(* IEC 61131-3 sources: LLM-CodeGen-TestGen/Tests, 13 files *)

(* ---- CRC_GEN.st ---- *)
FUNCTION_BLOCK CRC_GEN
  VAR_IN_OUT
    PT : ARRAY [0..249] OF BYTE;
  END_VAR
  VAR_INPUT
    SIZE : UINT;
    PL : UINT;
    PN : DWORD;
    INIT : DWORD;
    REV_IN : BOOL;
    REV_OUT : BOOL;
    XOR_OUT : DWORD;
  END_VAR
  VAR_OUTPUT
    _CRC_GEN : DWORD;
  END_VAR
  VAR
    pos : INT;
    shift : INT;
    bits : INT;
    dx : BYTE;
  END_VAR

  shift := 32 - UINT_TO_INT(PL);
  PN := SHL(PN, shift);

  (* load first 4 bytes into register minimum message size is 4 bytes
  	for smaller messages fill with 0#s at the beginning*)
  FOR pos := 0 TO 3 DO
  	IF REV_IN THEN _CRC_GEN := SHL(_CRC_GEN, 8) OR BYTE_TO_DWORD(REVERSE(PT[pos])); ELSE _CRC_GEN := SHL(_CRC_GEN, 8) OR BYTE_TO_DWORD(PT[pos]); END_IF;
  END_FOR;
  pos := 4;

  (* xor with init value *)
  _CRC_GEN := _CRC_GEN XOR SHL(init, shift);

  (* calculate CRC for each byte *)
  WHILE pos < UINT_TO_INT(size) DO
  	IF REV_IN THEN DX := REVERSE(PT[pos]); ELSE DX := PT[pos]; END_IF;
  	pos := pos + 1;
  	(* crc calculation for one byte *)
  	FOR bits := 0 TO 7 DO
  		IF (_CRC_GEN AND DWORD#16#8000_0000) > DWORD#0 THEN (* CRC_GEN.31 *)
  			_CRC_GEN := (SHL(_CRC_GEN, 1) OR BOOL_TO_DWORD((DX AND BYTE#16#80) > BYTE#0)) XOR PN; (* DX.7 *)
  		ELSE
  			_CRC_GEN := SHL(_CRC_GEN, 1) OR BOOL_TO_DWORD((DX AND BYTE#16#80) > BYTE#0); (* DX.7 *)
  		END_IF;
  		dx := SHL(dx, 1);
  	END_FOR;
  END_WHILE;

  (* all bytes are processed, need to finish the registers 32 bits *)
  FOR bits := 0 TO 31 DO
  	IF (_CRC_GEN AND DWORD#16#8000_0000) > DWORD#0 THEN (* CRC_GEN.31 *)
  		_CRC_GEN := (SHL(_CRC_GEN, 1) OR BOOL_TO_DWORD((DX AND BYTE#16#80) > BYTE#0)) XOR PN; (* DX.7 *)
  	ELSE
  		_CRC_GEN := SHL(_CRC_GEN, 1) OR BOOL_TO_DWORD((DX AND BYTE#16#80) > BYTE#0); (* DX.7 *)
  	END_IF;
  END_FOR;

  (* final XOR *)
  _CRC_GEN := SHR(_CRC_GEN, shift) XOR XOR_OUT;

  (* reverse the crc_out put if necessary *)
  IF REV_OUT THEN _CRC_GEN := REFLECT(_CRC_GEN, UINT_TO_INT(PL)); END_IF;

  (* typical crc polynoms

  CRC-4-ITU 			x4 + x + 1 					(ITU G.704, p. 12) 	0x3 or 0xC (0x9)
  CRC-5-ITU 			x5 + x4 + x2 + 1 			(ITU G.704, p. 9) 	0x15 or 0x15 (0x0B) Bluetooth
  CRC-5-USB 			x5 + x2 + 1 				(use: USB token packets) 	0x05 or 0x14 (0x9)
  CRC-6-ITU 			x6 + x + 1 					(ITU G.704, p. 3) 	0x03 or 0x30 (0x21)
  CRC-7 				x7 + x3 + 1 				(use: telecom systems, MMC) 	0x09 or 0x48 (0x11)
  CRC-8-ATM 			x8 + x2 + x + 1 				(use: ATM HEC) 	0x07 or 0xE0 (0xC1)
  CRC-8-CCITT 		x8 + x7 + x3 + x2 + 1 		(use: 1-Wire bus) 	0x8D or 0xB1 (0x63)
  CRC-8-Dallas/Maxim 	x8 + x5 + x4 + 1 			(use: 1-Wire bus) 	0x31 or 0x8C (0x19)
  CRC-8 				x8 + x7 + x6 + x4 + x2 + 1 	0xD5 or 0xAB (0x57)
  CRC-8-SAE J1850 	x8 + x4 + x3 + x2 + 1 		0x1D or 0xB8
  CRC-10 				x10 + x9 + x5 + x4 + x + 1 	0x233 or 0x331 (0x263)
  CRC-12 				x12 + x11 + x3 + x2 + x + 1 (use: telecom systems) 	0x80F or 0xF01 (0xE03)
  CRC-15-CAN 			x15 + x14 + x10 + x8 + x7 + x4 + x3 + 1 	0x4599 or 0x4CD1 (0x19A3)
  CRC-16-Fletcher 	Not a CRC; see Fletchers checksum 	Used in Adler-32 A & B CRCs
  CRC-16-CCITT 	x16 + x12 + x5 + 1 (XMODEM,X.25, V.41, Bluetooth, PPP, IrDA; known as "CRC-CCITT") 	0x1021 or 0x8408 (0x0811)
  CRC-16-IBM 	x16 + x15 + x2 + 1 (USB, many others; also known as "CRC-16") 	0x8005 or 0xA001 (0x4003)
  CRC-24-Radix-64 	x24 + x23 + x18 + x17 + x14 + x11 + x10 + x7 + x6 + x5 + x4 + x3 + x + 1 	0x864CFB or 0xDF3261 (0xBE64C3)
  CRC-32-Adler 	Not a CRC; see Adler-32 	See Adler-32
  CRC-32-MPEG2 	x32 + x26 + x23 + x22 + x16 + x12 + x11 + x10 + x8 + x7 + x5 + x4 + x2 + x + 1 	0x04C11DB7 or 0xEDB88320 (0xDB710641) Also used in IEEE 802.3
  CRC-32-IEEE 802.3 	x32 + x26 + x23 + x22 + x16 + x12 + x11 + x10 + x8 + x7 + x5 + x4 + x2 + x + 1 (V.42) 	0x04C11DB7 or 0xEDB88320 (0xDB710641)
  CRC-32C (Castagnoli) 	x32 + x28 + x27 + x26 + x25 + x23 + x22 + x20 + x19 + x18 + x14 + x13 + x11 + x10 + x9 + x8 + x6 + 1 	0x1EDC6F41 or 0x82F63B78 (0x05EC76F1)
  CRC-64-ISO 	x64 + x4 + x3 + x + 1 (use: ISO 3309) 	0x000000000000001B or 0xD800000000000000 (0xB000000000000001)
  CRC-64-ECMA-182 	x64 + x62 + x57 + x55 + x54 + x53 + x52 + x47 + x46 + x45 + x40 + x39 + x38 + x37 + x35 + x33 + x32 + x31 + x29 + x27 + x24 + x23 + x22 + x21 + x19 + x17 + x13 + x12 + x10 + x9 + x7 + x4 + x + 1
  (as described in ECMA-182 p.63) 	0x42F0E1EBA9EA3693 or 0xC96C5795D7870F42 (0x92D8AF2BAF0E1E85)
  *)
END_FUNCTION_BLOCK

(* ---- DEC_TO_HEX.st ---- *)
FUNCTION_BLOCK DEC_TO_HEX
  VAR_INPUT
    DecimalValue : DINT;
  END_VAR
  VAR_OUTPUT
    HexString : STRING;
  END_VAR
  VAR
    i : INT;
    hexDigits : ARRAY [0..15] OF STRING := ['0', '1', '2', '3', '4', '5', '6', '7', '8', '9', 'A', 'B', 'C', 'D', 'E', 'F'];
    digitIndex : INT;
    hexDigit : STRING;
    significantDigitFound : BOOL := FALSE;
    digitValue : DINT;
    powerOfInteger : DINT;
  END_VAR

  HexString := '';

  IF DecimalValue = 0 THEN
      HexString := '0';
      RETURN;
  END_IF;

  significantDigitFound := FALSE;

  FOR digitIndex := 0 TO 7 DO

      powerOfInteger:=1;
      FOR i := 1 TO 7 - digitIndex DO
        powerOfInteger := powerOfInteger * 16;
      END_FOR;

      digitValue := DIV(DecimalValue, powerOfInteger) MOD 16;
      hexDigit := hexDigits[digitValue];

      IF hexDigit <> '0' OR significantDigitFound OR (7 - digitIndex) = 0 THEN
          significantDigitFound := TRUE;
          HexString := CONCAT(HexString, hexDigit);
      END_IF;

  END_FOR;
END_FUNCTION_BLOCK

(* ---- FLOW_METER.st ---- *)
FUNCTION_BLOCK FLOW_METER
  VAR_INPUT
    VX : REAL;
    _E : BOOL;
    RST : BOOL;
    PULSE_MODE : BOOL;
    UPDATE_TIME : TIME := t#1s;
  END_VAR
  VAR_OUTPUT
    F : REAL;
  END_VAR
  VAR_IN_OUT
    X : REAL;
    Y : UDINT;
  END_VAR
  VAR
    tx : TIME;
    tl : TIME;
    int1 : INTEGRATE;
    init : BOOL;
    e_last : BOOL;
    tmp : INT;
    x_last : REAL;
    y_last : UDINT;
  END_VAR

  IF NOT init THEN	(* init on power up *)
  	init := TRUE;
  	tl := tx;
  	x_last := X;
  	y_last := Y;
  	int1.K := 2.7777777777777777E-4;
  END_IF;

  (* run integrator *)
  int1(_E := NOT (RST OR PULSE_MODE) AND _E, X := VX, Y := X);	(* gated operation *)
  X := int1.Y;

  IF RST THEN		(* reset *)
  	X := 0.0;
  	Y := UDINT#0;
  	tl := tx;
  	x_last := 0.0;
  	y_last := UDINT#0;
  ELSIF _E AND PULSE_MODE THEN	(* check for pulse mode *)
  	IF NOT e_last THEN X := X + VX; END_IF;
  END_IF;
  e_last := _E;

  (* reduce X to be less than 1 and increase Y respectively *)
  IF X > 1.0 THEN
  	tmp := FLOOR(X);
  	Y := Y + INT_TO_UDINT(tmp);
  	X := X - INT_TO_REAL(tmp);
  END_IF;

  (* calculate the current flow *)
  tx := UDINT_TO_TIME(T_PLC_MS(en:=true));
  IF tx - tl >= UPDATE_TIME AND UPDATE_TIME > t#0s THEN
  	F := (UDINT_TO_REAL(Y - y_last) + X - x_last) / TIME_TO_REAL(tx - tl) * 3.6E6;
  	y_last := Y;
  	x_last := X;
  	tl := tx;
  END_IF;

  (* From OSCAT Library, www.oscat.de *)
  (* T_PLC_MS, FLOOR, INTEGRATE required *)
END_FUNCTION_BLOCK

(* ---- FT_PIDWL.st ---- *)
FUNCTION_BLOCK FT_PIDWL
  VAR_INPUT
    IN : REAL;
    KP : REAL := 1.0;
    TN : REAL := 1.0;
    TV : REAL := 1.0;
    LIM_L : REAL := -1.0E38;
    LIM_H : REAL := 1.0E38;
    RST : BOOL;
  END_VAR
  VAR_OUTPUT
    Y : REAL;
    LIM : BOOL;
  END_VAR
  VAR
    piwl : FT_PIWL;
    diff : FT_DERIV;
  END_VAR

  IF rst THEN
  	piwl(rst := TRUE);
  	piwl.RST := FALSE;
  ELSE
  	(* run PIWL controller first *)
  	(* we need to check if TN = 0 and do alternative calls *)
  	IF TN = 0.0 THEN
  		piwl(in := IN * KP, KP := 1.0, KI := 0.0, LIM_L := LIM_L, LIM_H := LIM_H);
  	ELSE
  		piwl(in := IN * KP, KP := 1.0, KI := 1.0 / TN, LIM_L := LIM_L, LIM_H := LIM_H);
  	END_IF;

  	(* run differentiator and add_to_output *)
  	diff(IN := IN, K := KP * TV);
  	Y := piwl.Y + diff.out;

  	(* limit the output *)
  	IF Y < LIM_L THEN
  		LIM := TRUE;
  		Y := LIM_L;
  	ELSIF Y > LIM_H THEN
  		LIM := TRUE;
  		Y := LIM_H;
  	ELSE
  		LIM := FALSE;
  	END_IF;
  END_IF;

  (* From OSCAT Library, www.oscat.de *)
  (* T_PLC_US, FT_DERIV required *)
END_FUNCTION_BLOCK

(* ---- GEN_BIT.st ---- *)
FUNCTION_BLOCK GEN_BIT
  VAR_INPUT
    IN0 : DWORD;
    IN1 : DWORD;
    IN2 : DWORD;
    IN3 : DWORD;
    CLK : BOOL;
    STEPS : INT;
    REP : INT;
    RST : BOOL;
  END_VAR
  VAR_OUTPUT
    Q0 : BOOL;
    Q1 : BOOL;
    Q2 : BOOL;
    Q3 : BOOL;
    CNT : INT;
    RUN : BOOL;
  END_VAR
  VAR
    r0 : DWORD;
    r1 : DWORD;
    r2 : DWORD;
    r3 : DWORD;
    rx : INT := 1;
  END_VAR

  (* check if number of runs is finished or rep = 0 which means continuous *)

  IF clk AND NOT rst THEN
  	run := (rep = 0) OR (rx <= rep);
  	IF run THEN
  		(* check for step counter reached and reset to 0 if cnt = steps *)
  		IF cnt = steps THEN
  			cnt := 0;
  		END_IF;

  		(* when cnt = 0 then reload the inputs into the registers *)
  		IF cnt = 0 THEN
  			r0 := in0;
  			r1 := in1;
  			r2 := in2;
  			r3 := in3;
  		END_IF;

  		(* when cnt < steps, shift the lowest bits to the outputs *)
  		IF (cnt < steps) THEN
              Q0 := BIT_OF_DWORD(r0,0); (* Q0 := r0.X0; *)
              Q1 := BIT_OF_DWORD(r1,0); (* Q1 := r1.X0; *)
              Q2 := BIT_OF_DWORD(r2,0); (* Q2 := r2.X0; *)
              Q3 := BIT_OF_DWORD(r3,0); (* Q3 := r3.X0; *)
  			r0 := SHR(r0,1);
  			r1 := SHR(r1,1);
  			r2 := SHR(r2,1);
  			r3 := SHR(r3,1);
  		END_IF;

  		(* increment the step counter *)
  		cnt := cnt +1;
  		IF (cnt = steps) AND (rep <> 0) THEN rx := rx +1; END_IF;
  		IF (rx > rep) AND (rep <> 0) THEN run := FALSE; END_IF;
  	END_IF;
  ELSE
  	IF rst THEN
  		run := FALSE;
  		Q0 := FALSE;
  		Q1 := FALSE;
  		Q2 := FALSE;
  		Q3 := FALSE;
  		r0 := DWORD#0;
  		r1 := DWORD#0;
  		r2 := DWORD#0;
  		r3 := DWORD#0;
  		cnt := 0;
  		rx := 1;
  	END_IF;
  END_IF;

  (*From OSCAT Library, www.oscat.de *)
END_FUNCTION_BLOCK

(* ---- GEN_SIN.st ---- *)
FUNCTION_BLOCK GEN_SIN
  VAR_INPUT
    PT : TIME;
    AM : REAL := 1.0;
    OS : REAL;
    DL : REAL;
  END_VAR
  VAR_OUTPUT
    Q : BOOL;
    OUT : REAL;
  END_VAR
  VAR
    tx : TIME;
    last : TIME;
    init : BOOL;
    temp : REAL;
  END_VAR

  tx:= UDINT_TO_TIME(T_PLC_MS(en:=true)) - last;

  DL := modR(dl,1.0);
  IF dl < 0.0 THEN dl := 1.0 - dl; END_IF;

  (* init section *)
  IF NOT init THEN
  	init := TRUE;
  	last := tx;
  	tx := t#0s;
  END_IF;

  (* add last if one cycle is finished *)
  IF tx >= pt THEN
  	last := last + pt;
  	tx := tx - pt;
  END_IF;

  (* generate sine wave *)
  IF pt > t#0s THEN temp := SIN(6.283185307179586476 * TIME_TO_REAL(tx + multime(pt, dl)) / TIME_TO_REAL(pt)); END_IF;
  out := am * 0.5 *  temp + os;

  (* boolean output Q *)
  q := NOT sign_R(temp);

  (* From OSCAT Library, www.oscat.de *)
  (* T_PLC_MS, SIGN_R required*)
END_FUNCTION_BLOCK

(* ---- INCLUDE.st ---- *)
FUNCTION BIT_OF_DWORD : BOOL
  VAR_INPUT
    IN : DWORD;
    N : INT;
  END_VAR

  BIT_OF_DWORD := (SHR(in,N) AND 16#00000001) > 0;
  (* from OSCAT library; www.oscat.de  *)
END_FUNCTION

FUNCTION SIGN_R : BOOL
  VAR_INPUT
    IN : REAL;
  END_VAR

  SIGN_R := in < 0.0;
  (* from OSCAT library; www.oscat.de  *)
END_FUNCTION

FUNCTION FLOOR : INT
  VAR_INPUT
    x : REAL;
  END_VAR

  FLOOR := REAL_TO_INT(X);
  IF INT_TO_REAL(FLOOR) > X THEN
  	floor := floor - 1;
  END_IF;
  (* from OSCAT library; www.oscat.de  *)
END_FUNCTION

FUNCTION FLOOR2 : DINT
  VAR_INPUT
    x : REAL;
  END_VAR

  FLOOR2 := REAL_TO_DINT(X);
  IF DINT_TO_REAL(FLOOR2) > X THEN
  	FLOOR2 := FLOOR2 - DINT#1;
  END_IF;
  (* from OSCAT library; www.oscat.de  *)
END_FUNCTION

FUNCTION MODR : REAL
  VAR_INPUT
    IN : REAL;
    DIVI : REAL;
  END_VAR

  IF divi = 0.0 THEN
  	MODR := 0.0;
  ELSE
  	MODR := in - DINT_TO_REAL(FLOOR2(in / divi)) * divi;
  END_IF;
  (* from OSCAT library; www.oscat.de  *)
  (* FC FLOOR2 required *)
END_FUNCTION

FUNCTION REVERSE : BYTE
  VAR_INPUT
    IN : BYTE;
  END_VAR

  reverse := SHL(in,7) OR SHR(in,7) OR (ROR(in,3) AND BYTE#2#01000100) OR (ROL(in,3) AND BYTE#2#00100010)
  	OR (SHL(in,1) AND BYTE#2#00010000) OR (SHR(in,1) AND BYTE#2#00001000);

  (* Fromm Oscat Library, www.oscat.de *)
END_FUNCTION

FUNCTION REFLECT : DWORD
  VAR_INPUT
    DI : DWORD;
    L : INT;
  END_VAR
  VAR
    i : INT;
    _d : DWORD;
  END_VAR

  _d := DI;
  FOR i := 1 TO L DO
  	REFLECT := SHL(REFLECT, 1) OR BOOL_TO_DWORD((_d AND DWORD#2#0000_0001) > DWORD#0); (* D.0 *)
  	_d := SHR(_d, 1);
  END_FOR;
  REFLECT := REFLECT OR SHL(_d, L);

  (* Fromm Oscat Library, www.oscat.de *)
END_FUNCTION

FUNCTION BIT_LOAD_B : BYTE
  VAR_INPUT
    IN : BYTE;
    VAL : BOOL;
    POS : INT;
  END_VAR

  IF VAL THEN
  	BIT_LOAD_B := in OR SHL(BYTE#1,pos);
  ELSE
  	BIT_LOAD_B := in AND (NOT SHL(BYTE#1,pos));
  END_IF;

  (*From OSCAT Library, www.oscat.de*)
END_FUNCTION

FUNCTION _BYTE_TO_INT : INT
  VAR_INPUT
    IN : BYTE;
  END_VAR

  _BYTE_TO_INT := USINT_TO_INT(BYTE_TO_USINT(IN));

  (*From OSCAT Library, www.oscat.de*)
END_FUNCTION

FUNCTION T_PLC_MS : UDINT
  VAR
    tx : UDINT;
  END_VAR
  VAR_INPUT
    debug : BOOL;
  END_VAR
  VAR
    N : INT := 0;
    offset : UDINT := 0;
    temp : DWORD := 1;
  END_VAR

  tx := 0;
  {extern unsigned long __tick;
  extern unsigned long long common_ticktime__;
  unsigned long long ticktime_ms = (common_ticktime__)/1000000;
  UDINT plc_time = (UDINT)(ticktime_ms * (unsigned long long)__tick);
  TX = plc_time}
  T_PLC_MS := tx;
  IF debug THEN
  	T_PLC_MS := (DWORD_TO_UDINT(SHL(UDINT_TO_DWORD(T_PLC_MS),N) OR SHL(temp,N))-1) + OFFSET;
  END_IF;

  IF debug THEN
  	T_PLC_MS := (DWORD_TO_UDINT(SHL(UDINT_TO_DWORD(T_PLC_MS),N) OR SHL(temp,N))-1) + OFFSET;
  END_IF;

  (* Original Code:
  tx := TIME();
  T_PLC_MS := TIME_TO_DWORD(Tx);
  IF debug THEN
  	T_PLC_MS := (SHL(T_PLC_MS,N) OR SHL(DWORD#1,N)-1) + OFFSET;
  END_IF;
  *)

  (* From OSCAT library, www.oscat.de

  this is a temporary T_PLC_MS FB until OpenPLC gets it´s own time() functionality *)

  (* PLC_TIME and Global variables PLC_SCAN_CYCL and PLC_CYCL_TIME required *)
END_FUNCTION

FUNCTION T_PLC_US : UDINT
  VAR
    tx : UDINT;
  END_VAR
  VAR_INPUT
    debug : BOOL;
  END_VAR
  VAR
    N : INT := 0;
    offset : UDINT := 0;
    temp : DWORD := 1;
  END_VAR

  T_PLC_US := tx*1000;
  IF debug THEN
  	T_PLC_US := (DWORD_TO_UDINT(SHL(UDINT_TO_DWORD(T_PLC_US),N) OR SHL(temp,N))-1) + OFFSET;
  END_IF;

  (* Original Code:
  tx := TIME();
  T_PLC_US := TIME_TO_DWORD(Tx)*1000;
  IF debug THEN
  	T_PLC_US := (SHL(T_PLC_US,N) OR SHL(DWORD#1,N)-1) + OFFSET;
  END_IF;
  *)

  (* From OSCAT library, www.oscat.de

  this is a temporary T_PLC_US FB until OpenPLC gets it´s own time() functionality *)

  (* PLC_TIME and Global variables PLC_SCAN_CYCL and PLC_CYCL_TIME required *)
END_FUNCTION

FUNCTION_BLOCK FT_DERIV
  VAR_INPUT
    IN : REAL;
    K : REAL := 1.0;
    RUN : BOOL := TRUE;
  END_VAR
  VAR_OUTPUT
    OUT : REAL;
  END_VAR
  VAR
    old : REAL;
    tx : UDINT;
    last : UDINT;
    init : BOOL;
    tc : REAL;
  END_VAR

  tx:= T_PLC_US(en:=true);
  tc := UDINT_TO_REAL(tx - last);

  (* init on firsat startup *)
  IF NOT init THEN
  	init := TRUE;
  	old := in;
  ELSIF run AND tc > 0.0 THEN
  	out := (in - old) / tc * 1000000.0 * K;
  	old := in;
  ELSE
  	out := 0.0;
  END_IF;

  last := tx;

  (* From OSCAT Library, www.oscat.de *)
  (* T_PLC_US, required *)
END_FUNCTION_BLOCK

FUNCTION_BLOCK FT_PIWL
  VAR_INPUT
    IN : REAL;
    KP : REAL := 1.0;
    KI : REAL := 1.0;
    LIM_L : REAL := -1.0E38;
    LIM_H : REAL := 1.0E38;
    RST : BOOL;
  END_VAR
  VAR_OUTPUT
    Y : REAL;
    LIM : BOOL;
  END_VAR
  VAR
    init : BOOL;
    tx : UDINT;
    tc : REAL;
    t_last : UDINT;
    in_last : REAL;
    i : REAL;
    p : REAL;
  END_VAR

  IF NOT init OR RST THEN
  	init := TRUE;
  	in_last := in;
  		t_last := T_PLC_US(en:=true);
  	i := 0.0;
  	tc := 0.0;
  ELSE
  	(* read last cycle time in Microseconds *)
  		tx := T_PLC_US(en:=true);
  	tc := UDINT_TO_REAL(tx - t_last);
  	t_last := tx;

  	(* calculate proportional part *)
  	p := KP * IN;

  	(* run integrator *)
  	i := (IN + in_last) * 5.0E-7 * KI * tc + i;
  	in_last := IN;

  	(* calculate output Y *)
  	Y := p + i;

  	(* check output for limits *)
  	IF Y >= LIM_H THEN
  		Y := LIM_H;
  		IF ki <> 0.0 THEN
  			i := LIM_H - p;
  		ELSE
  			i := 0.0;
  		END_IF;
  		LIM := TRUE;
  	ELSIF Y <= LIM_L THEN
  		Y := LIM_L;
  		IF ki <> 0.0 THEN
  			i := LIM_L - p;
  		ELSE
  			i := 0.0;
  		END_IF;
  		LIM := TRUE;
  	ELSE
  		LIM := FALSE;
  	END_IF;
  END_IF;

  (* From OSCAT Library, www.oscat.de *)
  (* T_PLC_US required *)
END_FUNCTION_BLOCK

FUNCTION_BLOCK INTEGRATE
  VAR_INPUT
    _E : BOOL := TRUE;
    X : REAL;
    K : REAL := 1.0;
  END_VAR
  VAR_IN_OUT
    Y : REAL;
  END_VAR
  VAR
    x_last : REAL;
    init : BOOL;
    last : UDINT;
    tx : UDINT;
  END_VAR

  tx:= T_PLC_MS(en:=true);

  IF NOT init THEN
  	init := TRUE;
  	X_last := X;
  ELSIF _E THEN
  	Y := (X + X_LAST) * 0.5E-3 * UDINT_TO_REAL(tx-last) * K + Y;
  	X_last := X;
  END_IF;
  last := tx;

  (* From OSCAT Library, www.oscat.de *)
  (* T_PLC_MS required *)
END_FUNCTION_BLOCK

(* ---- LAMBERT_W.st ---- *)
FUNCTION_BLOCK LAMBERT_W
  VAR_INPUT
    X : REAL;
  END_VAR
  VAR_OUTPUT
    OUT : REAL;
  END_VAR
  VAR
    w : REAL;
    i : INT;
    we : REAL;
    w1e : REAL;
    ewx : REAL;
    last : DWORD;
  END_VAR

  IF x < -0.367879441171442 THEN
  	OUT := -1000.0;
  	RETURN;
  (* return 0 if x = 0 *)
  ELSIF x = 0.0 THEN
  	RETURN;
  (* first an estimate is calculated *)
  ELSIF x <= 500.0 THEN
  	w := LN(x + 1.0);
  	w := 0.665 * (1.0 + 0.0195 * w) * w + 0.04;
  ELSE
  	w := LN(x - 4.0) - (1.0 - 1.0/LN(x)) * LN(LN(x));
  END_IF;
  (* use estimate to calculate exact result *)
  FOR i := 0 TO 5 DO
  	ewx := EXP(w);
  	we := w * ewx - x;
  	w1e := (w+1.0) * ewx;
  	last := REAL_TO_DWORD(w) AND DWORD#16#FFFF_FFFC;
  	w := w - (we / (w1e - (w+2.0) * we / (2.0 * w + 2.0)));
  	IF (REAL_TO_DWORD(w) AND DWORD#16#FFFF_FFFC) = last THEN EXIT; END_IF;
  END_FOR;
  OUT := w;
  (* from OSCAT library; www.oscat.de  *)
END_FUNCTION_BLOCK

(* ---- MATRIX.st ---- *)
FUNCTION_BLOCK MATRIX
  VAR_INPUT
    X1 : BOOL;
    X2 : BOOL;
    X3 : BOOL;
    X4 : BOOL;
    X5 : BOOL;
    RELEASE : BOOL;
  END_VAR
  VAR_OUTPUT
    CODE : BYTE;
    _TP : BOOL;
    Y1 : BOOL := TRUE;
    Y2 : BOOL;
    Y3 : BOOL;
    Y4 : BOOL;
  END_VAR
  VAR
    line : BYTE;
    x : ARRAY [0..3] OF BYTE;
    l : ARRAY [0..3] OF BYTE;
    i : INT;
    temp : BYTE;
    temp2 : BYTE;
    L_temp : BYTE;
    temp_bit : BOOL;
    in_temp : INT;
  END_VAR

  _TP := FALSE;
  code := BYTE#0;

  (* read scan lines *)
  in_temp := _BYTE_TO_INT(line);
  temp := X[in_temp];  (* X[LINE] umkopieren *)

  temp:=BIT_LOAD_B(temp,X1,0); (* X[line].0 := X1; *)
  temp:=BIT_LOAD_B(temp,X2,1); (* X[line].1 := X2; *)
  temp:=BIT_LOAD_B(temp,X3,2); (* X[line].2 := X3; *)
  temp:=BIT_LOAD_B(temp,X4,3); (* X[line].3 := X4; *)
  temp:=BIT_LOAD_B(temp,X5,4); (* X[line].4 := X5; *)

  X[in_temp] := temp; (* X[LINE] zurückkopieren *)

  (* compare for change *)
  FOR i := 0 TO 3 DO
  	IF X[i] <> L[i] THEN
  		(* scan line information has changed code need to be found and generated *)
  		temp   := x[i] XOR L[i];
          temp2  := X[i];
          L_temp := L[i];

          IF BIT_OF_DWORD(BYTE_TO_DWORD(temp),0) THEN (* temp.l *)
  			code := BYTE#1;
              temp_bit := BIT_OF_DWORD(BYTE_TO_DWORD(temp2),0);   (* X[i].l *)
              code := BIT_LOAD_B(code,temp_bit,7);     			(* code.X7 *)
              L_temp := BIT_LOAD_B(L_temp,temp_bit,0); 			(* L[i].l *)
  		ELSIF BIT_OF_DWORD(BYTE_TO_DWORD(temp),1) THEN          (* temp.X1 *)
  			code := BYTE#2;
              temp_bit := BIT_OF_DWORD(BYTE_TO_DWORD(temp2),1);   (* X[i].X1 *)
              code := BIT_LOAD_B(code,temp_bit,7);     			(* code.X7 *)
              L_temp := BIT_LOAD_B(L_temp,temp_bit,1); 			(* L[i].X1 *)
  		ELSIF BIT_OF_DWORD(BYTE_TO_DWORD(temp),2) THEN          (* temp.X2 *)
  			code := BYTE#3;
              temp_bit := BIT_OF_DWORD(BYTE_TO_DWORD(temp2),2);   (* X[i].X2 *)
              code := BIT_LOAD_B(code,temp_bit,7);     			(* code.X7 *)
              L_temp := BIT_LOAD_B(L_temp,temp_bit,2); 			(* L[i].X2 *)
  		ELSIF BIT_OF_DWORD(BYTE_TO_DWORD(temp),3) THEN          (* temp.X3 *)
  			code := BYTE#4;
              temp_bit := BIT_OF_DWORD(BYTE_TO_DWORD(temp2),3);   (* X[i].X3 *)
              code := BIT_LOAD_B(code,temp_bit,7);     			(* code.X7 *)
              L_temp := BIT_LOAD_B(L_temp,temp_bit,3); 			(* L[i].X3 *)
  		ELSIF BIT_OF_DWORD(BYTE_TO_DWORD(temp),4) THEN          (* temp.X4 *)
  			code := BYTE#5;
              temp_bit := BIT_OF_DWORD(BYTE_TO_DWORD(temp2),4);   (* X[i].X4 *)
              code := BIT_LOAD_B(code,temp_bit,7);     			(* code.X7 *)
              L_temp := BIT_LOAD_B(L_temp,temp_bit,4); 			(* L[i].X4 *)
  		END_IF;
          L[i] := L_temp;
  		_TP := TRUE;
          code := (code AND BYTE#2#1000_1111) OR SHL(LINE AND BYTE#2#0000_0111,4);
          (* obere zeile enspricht: Code.X4 := Line.l; /  Code.X5 := Line.X1; / Code.RELEASE := Line.X2; *)

  		(* check if release codes need to be killed *)
  		IF NOT release AND code < BYTE#127 THEN
  			code := BYTE#0;
  			_TP := FALSE;
  		END_IF;
          EXIT;
  	END_IF;
  END_FOR;

  (* increment scan line every cycle *)
  line := INT_TO_BYTE(_BYTE_TO_INT(line) + 1) AND BYTE#2#0000_0011;
  temp := SHL(BYTE#1,_BYTE_TO_INT(line));

  Y1 := BIT_OF_DWORD(BYTE_TO_DWORD(temp),0); (* temp.0 *)
  Y2 := BIT_OF_DWORD(BYTE_TO_DWORD(temp),1); (* temp.1 *)
  Y3 := BIT_OF_DWORD(BYTE_TO_DWORD(temp),2); (* temp.2 *)
  Y4 := BIT_OF_DWORD(BYTE_TO_DWORD(temp),3); (* temp.3 *)

  (* Fromm Oscat Library, www.oscat.de *)
END_FUNCTION_BLOCK

(* ---- SEQUENCE_8.st ---- *)
FUNCTION_BLOCK SEQUENCE_8
  VAR_INPUT
    IN0 : BOOL := TRUE;
    IN1 : BOOL := TRUE;
    IN2 : BOOL := TRUE;
    IN3 : BOOL := TRUE;
    IN4 : BOOL := TRUE;
    IN5 : BOOL := TRUE;
    IN6 : BOOL := TRUE;
    IN7 : BOOL := TRUE;
    START : BOOL;
    RST : BOOL;
    WAIT0 : TIME;
    DELAY0 : TIME;
    WAIT1 : TIME;
    DELAY1 : TIME;
    WAIT2 : TIME;
    DELAY2 : TIME;
    WAIT3 : TIME;
    DELAY3 : TIME;
    WAIT4 : TIME;
    DELAY4 : TIME;
    WAIT5 : TIME;
    DELAY5 : TIME;
    WAIT6 : TIME;
    DELAY6 : TIME;
    WAIT7 : TIME;
    DELAY7 : TIME;
    STOP_ON_ERROR : BOOL;
  END_VAR
  VAR_OUTPUT
    Q0 : BOOL;
    Q1 : BOOL;
    Q2 : BOOL;
    Q3 : BOOL;
    Q4 : BOOL;
    Q5 : BOOL;
    Q6 : BOOL;
    Q7 : BOOL;
    QX : BOOL;
    RUN : BOOL;
    _STEP : INT := -1;
    STATUS : BYTE;
  END_VAR
  VAR
    last : TIME;
    edge : BOOL;
    tx : TIME;
    init : BOOL;
  END_VAR

  tx:= UDINT_TO_TIME(T_PLC_MS(en:=true));

  (* initialize on startup *)
  IF NOT init THEN
  	last := tx;
  	init := TRUE;
  	status := BYTE#110;
  END_IF;

  (* asynchronous reset *)
  IF rst THEN
  	_step := -1;
  	Q0 := FALSE;
  	Q1 := FALSE;
  	Q2 := FALSE;
  	Q3 := FALSE;
  	Q4 := FALSE;
  	Q5 := FALSE;
  	Q6 := FALSE;
  	Q7 := FALSE;
  	status := BYTE#110;
  	run := FALSE;

  (* edge on start input restarts the sequencer *)
  ELSIF start AND NOT edge THEN
  	_step := 0;
  	last := tx;
  	status := BYTE#111;
  	Q0 := FALSE;
  	Q1 := FALSE;
  	Q2 := FALSE;
  	Q3 := FALSE;
  	Q4 := FALSE;
  	Q5 := FALSE;
  	Q6 := FALSE;
  	Q7 := FALSE;
  	run := TRUE;
  END_IF;
  edge := start;

  (* check if stop on error is necessary *)
  IF status > BYTE#0 AND status < BYTE#100 AND stop_on_error THEN RETURN; END_IF;

  (* sequence is running *)
  IF run AND _step = 0 THEN
  	IF NOT q0 AND in0 AND tx - last <= wait0 THEN
  		Q0 := TRUE;
  		last := tx;
  	ELSIF NOT q0 AND tx - last > wait0 THEN
  		status := BYTE#1;
  		run := FALSE;
  	ELSIF q0 AND tx - last >= delay0 THEN
  		_step := 1;
  		last := tx;
  	END_IF;
  END_IF;
  IF run AND _step = 1 THEN
  	IF NOT q1 AND in1 AND tx - last <= wait1 THEN
  		Q0 := FALSE;
  		Q1 := TRUE;
  		last := tx;
  	ELSIF NOT q1 AND Tx - last > wait1 THEN
  		status := BYTE#2;
  		q0 := FALSE;
  		run := FALSE;
  	ELSIF q1 AND tx - last >= delay1 THEN
  		_step := 2;
  		last := tx;
  	END_IF;
  END_IF;
  IF run AND _step = 2 THEN
  	IF NOT q2 AND in2 AND tx - last <= wait2 THEN
  		Q1 := FALSE;
  		Q2 := TRUE;
  		last := tx;
  	ELSIF NOT q2 AND Tx - last > wait2 THEN
  		status := BYTE#3;
  		q1 := FALSE;
  		run := FALSE;
  	ELSIF q2 AND tx - last >= delay2 THEN
  		_step := 3;
  		last := tx;
  	END_IF;
  END_IF;
  IF run AND _step = 3 THEN
  	IF NOT q3 AND in3 AND tx - last <= wait3 THEN
  		Q2 := FALSE;
  		Q3 := TRUE;
  		last := tx;
  	ELSIF NOT q3 AND Tx - last > wait3 THEN
  		status := BYTE#4;
  		q2 := FALSE;
  		run := FALSE;
  	ELSIF q3 AND tx - last >= delay3 THEN
  		_step := 4;
  		last := tx;
  	END_IF;
  END_IF;
  IF run AND _step = 4 THEN
  	IF NOT q4 AND in4 AND tx - last <= wait4 THEN
  		Q3 := FALSE;
  		Q4 := TRUE;
  		last := tx;
  	ELSIF NOT q4 AND Tx - last > wait4 THEN
  		status := BYTE#5;
  		q3 := FALSE;
  		run := FALSE;
  	ELSIF q4 AND tx - last >= WAIT4 THEN
  		_step := 5;
  		last := tx;
  	END_IF;
  END_IF;
  IF run AND _step = 5 THEN
  	IF NOT q5 AND in5 AND tx - last <= DELAY4 THEN
  		Q4 := FALSE;
  		Q5 := TRUE;
  		last := tx;
  	ELSIF NOT q5 AND Tx - last > DELAY4 THEN
  		status := BYTE#6;
  		q4 := FALSE;
  		run := FALSE;
  	ELSIF q5 AND tx - last >= WAIT5 THEN
  		_step := 6;
  		last := tx;
  	END_IF;
  END_IF;
  IF run AND _step = 6 THEN
  	IF NOT q6 AND in6 AND tx - last <= DELAY5 THEN
  		Q5 := FALSE;
  		Q6 := TRUE;
  		last := tx;
  	ELSIF NOT q6 AND Tx - last > DELAY5 THEN
  		status := BYTE#7;
  		q5 := FALSE;
  		run := FALSE;
  	ELSIF q6 AND tx - last >= WAIT6 THEN
  		_step := 7;
  		last := tx;
  	END_IF;
  END_IF;
  IF run AND _step = 7 THEN
  	IF NOT q7 AND in7 AND tx - last <= DELAY6 THEN
  		Q6 := FALSE;
  		Q7 := TRUE;
  		last := tx;
  	ELSIF NOT q7 AND Tx - last > DELAY6 THEN
  		status := BYTE#8;
  		q6 := FALSE;
  		run := FALSE;
  	ELSIF q7 AND tx - last >= WAIT7 THEN
  		_step := -1;
  		Q7 := FALSE;
  		Run := FALSE;
  		status := BYTE#110;
  	END_IF;
  END_IF;
  QX := q0 OR q1 OR q2 OR q3 OR q4 OR q5 OR q6 OR q7;

  (*From OSCAT Library, www.oscat.de *)
END_FUNCTION_BLOCK

(* ---- TOOL_CHANGER.st ---- *)
FUNCTION_BLOCK TOOL_CHANGER

VAR_INPUT
    ToolChangeRequired : BOOL; (** True if tool change is required **)
    ToolCarouselPosition : INT; (** Current position of the tool carousel **)
    DesiredToolNumber : INT; (** Number of the desired tool **)
END_VAR

VAR_OUTPUT
    RotateCarousel : BOOL; (** Rotate the tool carousel **)
    LockTool : BOOL; (** Lock the tool in the spindle **)
END_VAR

VAR
    ToolChangeState : INT; (**0=Idle, 1=RotatingCarousel, 2=LockingTool**)
END_VAR

IF ToolChangeRequired THEN
    CASE ToolChangeState OF
        0:
            (** Check if carousel needs to rotate **)
            IF ToolCarouselPosition <> DesiredToolNumber THEN
                RotateCarousel := TRUE;
                ToolChangeState := 1;
            ELSE
                LockTool := TRUE;
                ToolChangeState := 2;
            END_IF;

        1:
            (** Wait for carousel to reach desired position **)
            IF ToolCarouselPosition = DesiredToolNumber THEN
                RotateCarousel := FALSE;
                LockTool := TRUE;
                ToolChangeState := 2;
            END_IF;

        2:
            (** Wait for tool to be locked **)
            LockTool := FALSE;
            ToolChangeState := 0;
    END_CASE;
END_IF;

END_FUNCTION_BLOCK

(* ---- TRAFFIC_CTRL.st ---- *)
FUNCTION_BLOCK TRAFFIC_CTRL

VAR_INPUT
    PedestrianButton1 : BOOL;
    PedestrianButton2 : BOOL;
END_VAR

VAR_OUTPUT
    NorthSouthRed : BOOL;
    NorthSouthYellow : BOOL;
    NorthSouthGreen : BOOL;
    EastWestRed : BOOL;
    EastWestYellow : BOOL;
    EastWestGreen : BOOL;
    PedestrianLight1 : BOOL;
    PedestrianLight2 : BOOL;
END_VAR

VAR
    LightState : INT := 0; (* 0: North-South Green, 1: North-South Yellow, 2: East-West Green, 3: East-West Yellow *)
    PedestrianRequest1 : BOOL := FALSE;
    PedestrianRequest2 : BOOL := FALSE;
    PedestrianCrossing : BOOL := FALSE;
    Timer : TON;
END_VAR

(* Check for pedestrian requests *)
IF PedestrianButton1 THEN
    PedestrianRequest1 := TRUE;
END_IF;

IF PedestrianButton2 THEN
    PedestrianRequest2 := TRUE;
END_IF;

(* Traffic light state machine *)
CASE LightState OF
    0: (* North-South Green *)
        NorthSouthGreen := TRUE;
        EastWestRed := TRUE;
        IF PedestrianRequest1 OR PedestrianRequest2 THEN
            Timer(IN := TRUE, PT := T#2s); (* Pedestrian crossing grace period *)
            IF Timer.Q THEN
                Timer(IN := FALSE);
                LightState := 1;
            END_IF;
        END_IF;

    1: (* North-South Yellow *)
        NorthSouthYellow := TRUE;
        EastWestRed := TRUE;
        Timer(IN := TRUE, PT := T#2s); (* Yellow light duration *)
        IF Timer.Q THEN
            Timer(IN := FALSE);
            LightState := 2;
        END_IF;

    2: (* East-West Green *)
        EastWestGreen := TRUE;
        NorthSouthRed := TRUE;
        IF PedestrianRequest1 THEN
            PedestrianLight1 := TRUE;
            PedestrianCrossing := TRUE;
        END_IF;
        IF PedestrianRequest2 THEN
            PedestrianLight2 := TRUE;
            PedestrianCrossing := TRUE;
        END_IF;
        IF PedestrianCrossing THEN
            Timer(IN := TRUE, PT := T#2s); (* Pedestrian crossing period *)
            IF Timer.Q THEN
                Timer(IN := FALSE);
                PedestrianRequest1 := FALSE;
                PedestrianRequest2 := FALSE;
                PedestrianLight1 := FALSE;
                PedestrianLight2 := FALSE;
                PedestrianCrossing := FALSE;
                LightState := 3;
            END_IF;
        END_IF;

    3: (* East-West Yellow *)
        EastWestYellow := TRUE;
        NorthSouthRed := TRUE;
        Timer(IN := TRUE, PT := T#2s); (* Yellow light duration *)
        IF Timer.Q THEN
            Timer(IN := FALSE);
            LightState := 0;
        END_IF;

END_CASE;

END_FUNCTION_BLOCK

(* ---- template.st ---- *)
CONFIGURATION Config0

  RESOURCE Res0 ON PLC
    TASK task0(INTERVAL := T#100ms,PRIORITY := 0);
    PROGRAM instance0 WITH task0 : TestRunnerProgram;
  END_RESOURCE
END_CONFIGURATION
